TYPE ST_DebugTcHmi :
STRUCT
	TestBool	: BOOL;
	TestInt		: UINT;
	TestLint	: ULINT;
END_STRUCT
END_TYPE

(* stored: Version 1.1.0.1
   DUT ST_DebugTcHmi: Id {33d77131-e73c-08cf-39b3-792dd0577710} *)
